GLOBALCONSTANTS DefaultPool (* Global constants *)
  VAR_GLOBAL CONSTANT
    ISO_DESIGNATOR_WIDTH : UINT := 80;
    ISO_DESIGNATOR_HEIGHT : UINT := 80;
    ISO_MASK_SIZE : UINT := 480;
    ISO_VERSION_LABEL : STRING;
    MASK_WIDTH : UINT := 480;
    MASK_HEIGHT : UINT := 480;
    WorkingSet_0 : UINT := 0;
    Macro_1 : UINT := 1;
    Macro_2 : UINT := 2;
    Macro_3 : UINT := 3;
    Macro_4 : UINT := 4;
    Macro_5 : UINT := 5;
    Macro_6 : UINT := 6;
    Macro_7 : UINT := 7;
    Macro_8 : UINT := 8;
    Macro_9 : UINT := 9;
    DataMask_M3 : UINT := 1000;
    DataMask_M4 : UINT := 1001;
    DataMask_M1 : UINT := 1002;
    DataMask_M2 : UINT := 1003;
    DataMask_M5 : UINT := 1004;
    Container_M1_weight : UINT := 3000;
    Container_M3_radar_speed : UINT := 3001;
    Container_M1_speed : UINT := 3002;
    Container_M3_wheel_speed : UINT := 3003;
    Container_W1_actual_quantity : UINT := 3004;
    Container_M1_percent : UINT := 3005;
    Container_M1_kg_ha : UINT := 3006;
    Container_M1_filllevel : UINT := 3007;
    Container_W1_flow_factor : UINT := 3008;
    Container_M1_electric_motor : UINT := 3009;
    Container_W1_target_quantity : UINT := 3010;
    Container_W1_engine_speed_percent : UINT := 3011;
    Container_W1_engine_speed_rpm : UINT := 3012;
    Container_M2_target_quantity : UINT := 3013;
    Container_W1_header : UINT := 3014;
    Container_M2_flow_factor : UINT := 3015;
    Container_M2_calibration_area : UINT := 3016;
    Container_Picture_fertilzier_bin_full_M1_filllevel : UINT := 3017;
    Container_Picture_fertilzier_bin_empty_M1_filllevel : UINT := 3018;
    SoftKeyMask_S1 : UINT := 4000;
    SoftKeyMask_S2 : UINT := 4001;
    SoftKeyMask_S3 : UINT := 4002;
    SoftKeyMask_S4 : UINT := 4003;
    SoftKey_stop : UINT := 5000;
    SoftKey_100_percent : UINT := 5001;
    SoftKey_plus_percent : UINT := 5002;
    SoftKey_start : UINT := 5003;
    SoftKey_minus_percent : UINT := 5004;
    SoftKey_main : UINT := 5005;
    SoftKey_debug : UINT := 5006;
    SoftKey_calibration_run : UINT := 5007;
    SoftKey_settings : UINT := 5008;
    SoftKey_5009 : UINT := 5009;
    SoftKey_5010 : UINT := 5010;
    SoftKey_5011 : UINT := 5011;
    SoftKey_5012 : UINT := 5012;
    SoftKey_5013 : UINT := 5013;
    SoftKey_5014 : UINT := 5014;
    SoftKey_5015 : UINT := 5015;
    SoftKey_5016 : UINT := 5016;
    SoftKey_5017 : UINT := 5017;
    SoftKey_5018 : UINT := 5018;
    SoftKey_5019 : UINT := 5019;
    SoftKey_5020 : UINT := 5020;
    SoftKey_5021 : UINT := 5021;
    SoftKey_5022 : UINT := 5022;
    SoftKey_5023 : UINT := 5023;
    SoftKey_5024 : UINT := 5024;
    SoftKey_5025 : UINT := 5025;
    SoftKey_5026 : UINT := 5026;
    SoftKey_5027 : UINT := 5027;
    Button_M1_reset : UINT := 6000;
    Button_M3_radar_speed_select : UINT := 6001;
    Button_M4_manuel_start : UINT := 6002;
    Button_M3_wheel_speed_select : UINT := 6003;
    Button_M4_manuel_stop : UINT := 6004;
    Button_6005 : UINT := 6005;
    Button_6006 : UINT := 6006;
    Button_W1_stop : UINT := 6007;
    Button_M1_refresh : UINT := 6008;
    Button_6009 : UINT := 6009;
    Button_M2_start : UINT := 6010;
    Button_M4_auto : UINT := 6011;
    Button_M2_calibration_area_1a : UINT := 6013;
    Button_M2_calibration_area_5a : UINT := 6014;
    Button_M2_calibration_area_10a : UINT := 6015;
    InputString_M4_P : UINT := 8000;
    InputString_M4_I : UINT := 8001;
    InputString_D : UINT := 8002;
    InputNumber_W1_actual_quantity : UINT := 9000;
    InputNumber_9001 : UINT := 9001;
    InputNumber_M2_target_quantity : UINT := 9002;
    InputNumber_M2_flow_factor : UINT := 9003;
    InputNumber_9004 : UINT := 9004;
    InputNumber_M4_motor_speed : UINT := 9005;
    InputNumber_M4_P : UINT := 9006;
    InputNumber_M4_I : UINT := 9007;
    InputNumber_M4_D : UINT := 9008;
    InputNumber_M4_auto : UINT := 9009;
    OutputString_M3_radar_speed_kmh : UINT := 11000;
    OutputString_M1_settings_header : UINT := 11001;
    OutputString_M1_kg_ha : UINT := 11002;
    OutputString_M1_filllevel : UINT := 11003;
    OutputString_W1_actual_quantity_g : UINT := 11004;
    OutputString_M3_radar_speed_header : UINT := 11005;
    OutputString_11006 : UINT := 11006;
    OutputString_M4_debug : UINT := 11007;
    OutputString_M1_header : UINT := 11008;
    OutputString_M2_header : UINT := 11009;
    OutputString_M1_reset : UINT := 11010;
    OutputString_M3_radar_speed_x : UINT := 11011;
    OutputString_SK_start : UINT := 11012;
    OutputString_SK_stop : UINT := 11013;
    OutputString_M1_weight : UINT := 11014;
    OutputString_M1_percent : UINT := 11015;
    OutputString_M1_electric_motor : UINT := 11016;
    OutputString_11017 : UINT := 11017;
    OutputString_M3_wheel_speed_kmh : UINT := 11018;
    OutputString_M3_wheel_speed_header : UINT := 11019;
    OutputString_M3_wheel_speed_x : UINT := 11020;
    OutputString_W1_actual_quantity_header : UINT := 11021;
    OutputString_W1_flow_factor : UINT := 11022;
    OutputString_W1_target_quantity : UINT := 11023;
    OutputString_W1_engine_speed_percent : UINT := 11024;
    OutputString_W1_engine_speed_rpm : UINT := 11025;
    OutputString_M2_target_quantity_kg : UINT := 11026;
    OutputString_W1_header : UINT := 11027;
    OutputString_W1_stop : UINT := 11028;
    OutputString_M2_target_quantity_header : UINT := 11029;
    OutputString_M2_start : UINT := 11030;
    OutputString_11031 : UINT := 11031;
    OutputString_M2_flow_factor_header : UINT := 11032;
    OutputString_M2_calibration_area : UINT := 11033;
    OutputString_M2_calibration_area_1a : UINT := 11034;
    OutputString_M2_calibration_area_5a : UINT := 11035;
    OutputString_M2_calibration_area_10a : UINT := 11036;
    OutputString_M4_manuel : UINT := 11037;
    OutputString_M4_engine_speed_manuel : UINT := 11038;
    OutputString_M4_auto : UINT := 11039;
    OutputString_11040 : UINT := 11040;
    OutputNumber_W1_flow_factor : UINT := 12000;
    OutputNumber_M3_radar_speed : UINT := 12002;
    OutputNumber_M1_speed : UINT := 12003;
    OutputNumber_M1_percent : UINT := 12004;
    OutputNumber_M1_weight : UINT := 12007;
    OutputNumber_M1_electric_motor : UINT := 12009;
    OutputNumber_M3_wheel_speed : UINT := 12010;
    OutputNumber_W1_target_quantity : UINT := 12011;
    OutputNumber_W1_engine_speed_percent : UINT := 12012;
    OutputNumber_W1_engine_speed_rpm : UINT := 12013;
    OutputNumber_12014 : UINT := 12014;
    Line_13000 : UINT := 13000;
    Rectangle_M1_percent : UINT := 14000;
    Rectangle_M1_speed : UINT := 14001;
    Rectangle_M1_kg_ha : UINT := 14002;
    Rectangle_M1_filllevel : UINT := 14003;
    Rectangle_M1_weight : UINT := 14004;
    Rectangle_M1_electric_motor : UINT := 14005;
    Rectangle_M3_radar_speed : UINT := 14007;
    Rectangle_M3_wheel_speed : UINT := 14008;
    Rectangle_M2_target_quantity : UINT := 14009;
    Rectangle_W1_actual_quantity : UINT := 14010;
    Rectangle_W1_flow_factor : UINT := 14011;
    Rectangle_W1_target_quantity : UINT := 14012;
    Rectangle_W1_engine_speed_percent : UINT := 14013;
    Rectangle_W1_engine_speed_rpm : UINT := 14014;
    Rectangle_W1_header : UINT := 14015;
    Rectangle_M2_flow_factor : UINT := 14016;
    Rectangle_M2_calibration_area : UINT := 14017;
    weight_W1_actual_quantity : UINT := 20000;
    _100_percent_softkeys : UINT := 20001;
    debug_softkeys : UINT := 20002;
    Tractor_ground_speed_M3_radar_speed : UINT := 20003;
    plus_percent_softkeys : UINT := 20004;
    minus_percent_softkeys : UINT := 20005;
    fertilzier_bin_softkeys : UINT := 20006;
    measuring_cup_softkeys : UINT := 20007;
    settings_softkeys : UINT := 20008;
    Picture_Tractor_forward_side_M1_speed : UINT := 20009;
    Picturere_Graphic_refresh : UINT := 20010;
    Picture_fertilzier_bin_empty_M1_filllevel : UINT := 20012;
    Picture_M1_weight : UINT := 20013;
    Picture_application_rate_per_area_M1_kg_ha : UINT := 20014;
    Picture_application_rate_per_area_M1_percent : UINT := 20015;
    Picture_fertilzier_bin_full_M1_filllevel : UINT := 20016;
    Picture_M1_electric_motor : UINT := 20018;
    Tractor_wheel_slip_M3_wheel_speed : UINT := 20021;
    fertilzier_bin_W1_flow_factor : UINT := 20026;
    weight_W1_target_quantity : UINT := 20028;
    Electric_motor_W1_engine_speed_percent : UINT := 20029;
    Electric_motor_W1_engine_speed_rpm : UINT := 20030;
    weight_20031 : UINT := 20031;
    application_rate_per_area_M2_target_quantity : UINT := 20037;
    application_rate_per_area_20039 : UINT := 20039;
    fertilzier_bin_M2_flow_factor : UINT := 20040;
    fertilzier_bin_20041 : UINT := 20041;
    NumberVariable_engine_speed_percent : UINT := 21000;
    NumberVariable_Ground_based_machine_speed : UINT := 21001;
    NumberVariable_bool_selected_speed : UINT := 21002;
    NumberVariable_target_quantity_calibration_run : UINT := 21003;
    NumberVariable_selected_speed : UINT := 21004;
    NumberVariable_engine_speed_manuel : UINT := 21005;
    NumberVariable_weight : UINT := 21006;
    NumberVariable_P : UINT := 21007;
    NumberVariable_application_rate_percent : UINT := 21008;
    NumberVariable_D : UINT := 21009;
    NumberVariable_manuel_auto_speed : UINT := 21010;
    NumberVariable_Wheel_based_machine_speed : UINT := 21011;
    NumberVariable_flow_factor_new : UINT := 21012;
    NumberVariable_target_quantity : UINT := 21013;
    NumberVariable_W1_actual_quantity : UINT := 21014;
    NumberVariable_engine_speed_rpm : UINT := 21015;
    NumberVariable_flow_factor : UINT := 21016;
    NumberVariable_I : UINT := 21017;
    NumberVariable_application_rate_percent_old : UINT := 21018;
    StringVariable_calibration_run : UINT := 22000;
    FontAttributes_23000 : UINT := 23000;
    FontAttributes_23001 : UINT := 23001;
    FontAttributes_Header : UINT := 23002;
    FontAttributes_WindowMask : UINT := 23003;
    FontAttributes_23005 : UINT := 23005;
    FontAttributes_23006 : UINT := 23006;
    FontAttributes_reset : UINT := 23009;
    FontAttributes_string_start_stop_button : UINT := 23010;
    FontAttributes_main_boxes : UINT := 23011;
    FontAttributes_23016 : UINT := 23016;
    FontAttributes_Header_white : UINT := 23018;
    LineAttributes_24000 : UINT := 24000;
    LineAttributes_24001 : UINT := 24001;
    LineAttributes_24002 : UINT := 24002;
    LineAttributes_24003 : UINT := 24003;
    LineAttributes_24004 : UINT := 24004;
    LineAttributes_24006 : UINT := 24006;
    LineAttributes_24007 : UINT := 24007;
    LineAttributes_24008 : UINT := 24008;
    LineAttributes_24009 : UINT := 24009;
    LineAttributes_24010 : UINT := 24010;
    LineAttributes_24011 : UINT := 24011;
    LineAttributes_24012 : UINT := 24012;
    LineAttributes_24013 : UINT := 24013;
    LineAttributes_24014 : UINT := 24014;
    LineAttributes_24015 : UINT := 24015;
    LineAttributes_24016 : UINT := 24016;
    FillAttributes_main_colour : UINT := 25011;
    FillAttributes_new_holland_blue : UINT := 25012;
  END_VAR
END_GLOBALCONSTANTS
